Staubli VAL3: read_ID.pgx

program read_ID()
begin
  do

    putln(getMoveId())
    ID_val = getMoveId()

  until check_ID != true
end
